INTERFACE Object

METHOD getNotification : STRING
VAR_INPUT
END_VAR
END_METHOD

END_INTERFACE

(* stored: Version 1.1.0.1, ProductVersion 3.1.4024.12
   Itf Object: Id {0988eda9-9fad-447e-bc17-ba4b26c3e534}
   Method getNotification: Id {947495b9-1c2e-4a6c-ad55-07922478da92} *)
